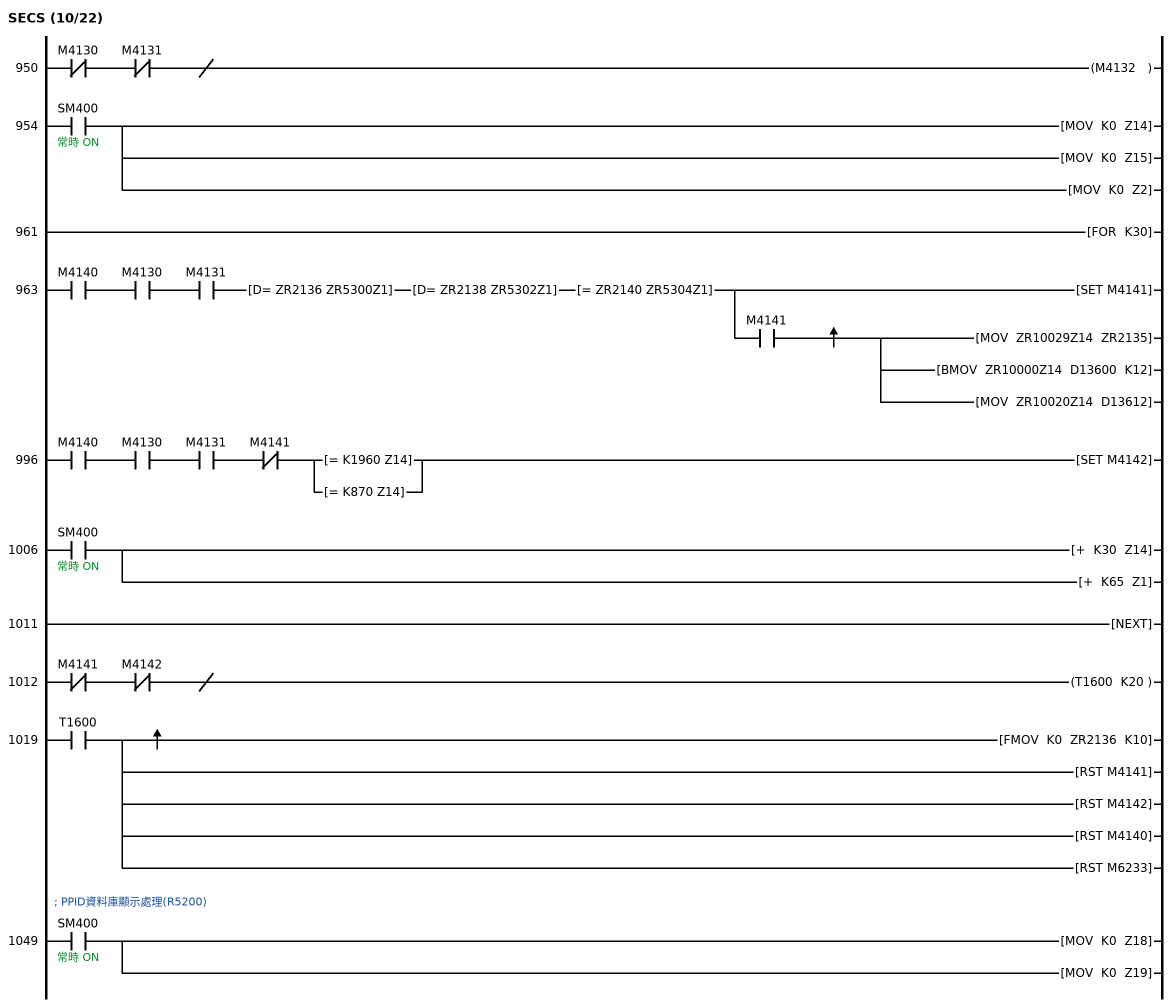
950   LDI     M4130
      ANI     M4131
      INV
      OUT     M4132
954   LD      SM400  ; 常時 ON
      MOV     K0 Z14
      MOV     K0 Z15
      MOV     K0 Z2
961   FOR     K30
963   LD      M4140
      AND     M4130
      AND     M4131
      ANDD=   ZR2136 ZR5300Z1
      ANDD=   ZR2138 ZR5302Z1
      AND=    ZR2140 ZR5304Z1
      SET     M4141
      AND     M4141
      MEP
      MOV     ZR10029Z14 ZR2135
      BMOV    ZR10000Z14 D13600 K12
      MOV     ZR10020Z14 D13612
996   LD      M4140
      AND     M4130
      AND     M4131
      ANI     M4141
      LD=     K1960 Z14
      OR=     K870 Z14
      ANB
      SET     M4142
1006  LD      SM400  ; 常時 ON
      +       K30 Z14
      +       K65 Z1
1011  NEXT
1012  LDI     M4141
      ANI     M4142
      INV
      OUT     T1600 K20
1019  LD      T1600
      MPS
      MEP
      FMOV    K0 ZR2136 K10
      MPP
      RST     M4141
      RST     M4142
      RST     M4140
      RST     M6233
; PPID資料庫顯示處理(R5200)
1049  LD      SM400  ; 常時 ON
      MOV     K0 Z18
      MOV     K0 Z19
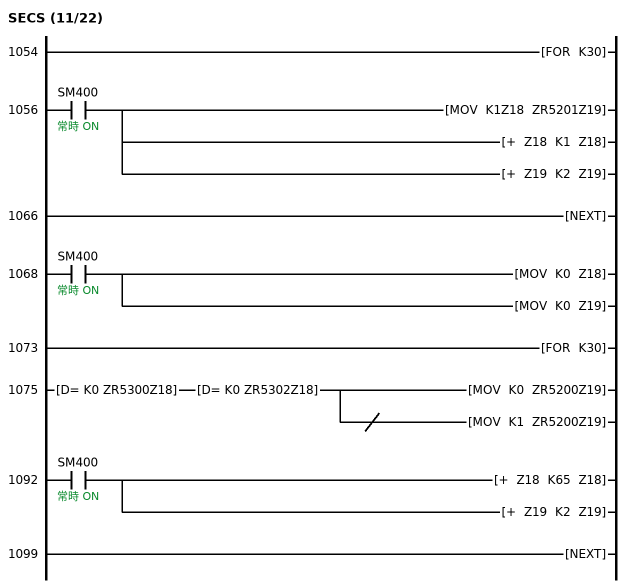
1054  FOR     K30
1056  LD      SM400  ; 常時 ON
      MOV     K1Z18 ZR5201Z19
      +       Z18 K1 Z18
      +       Z19 K2 Z19
1066  NEXT
1068  LD      SM400  ; 常時 ON
      MOV     K0 Z18
      MOV     K0 Z19
1073  FOR     K30
1075  LDD=    K0 ZR5300Z18
      ANDD=   K0 ZR5302Z18
      MOV     K0 ZR5200Z19
      INV
      MOV     K1 ZR5200Z19
1092  LD      SM400  ; 常時 ON
      +       Z18 K65 Z18
      +       Z19 K2 Z19
1099  NEXT
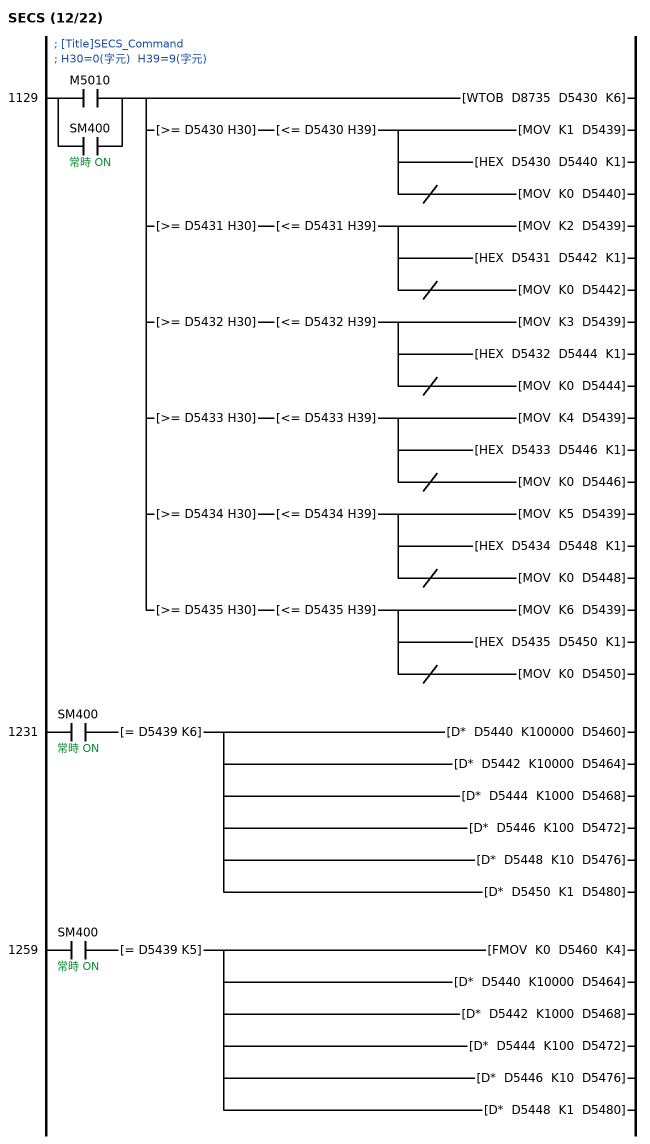
; [Title]SECS_Command
; H30=0(字元)  H39=9(字元)
1129  LD      M5010
      OR      SM400  ; 常時 ON
      WTOB    D8735 D5430 K6
      MPS
      AND>=   D5430 H30
      AND<=   D5430 H39
      MOV     K1 D5439
      HEX     D5430 D5440 K1
      INV
      MOV     K0 D5440
      MRD
      AND>=   D5431 H30
      AND<=   D5431 H39
      MOV     K2 D5439
      HEX     D5431 D5442 K1
      INV
      MOV     K0 D5442
      MRD
      AND>=   D5432 H30
      AND<=   D5432 H39
      MOV     K3 D5439
      HEX     D5432 D5444 K1
      INV
      MOV     K0 D5444
      MRD
      AND>=   D5433 H30
      AND<=   D5433 H39
      MOV     K4 D5439
      HEX     D5433 D5446 K1
      INV
      MOV     K0 D5446
      MRD
      AND>=   D5434 H30
      AND<=   D5434 H39
      MOV     K5 D5439
      HEX     D5434 D5448 K1
      INV
      MOV     K0 D5448
      MPP
      AND>=   D5435 H30
      AND<=   D5435 H39
      MOV     K6 D5439
      HEX     D5435 D5450 K1
      INV
      MOV     K0 D5450
1231  LD      SM400  ; 常時 ON
      AND=    D5439 K6
      D*      D5440 K100000 D5460
      D*      D5442 K10000 D5464
      D*      D5444 K1000 D5468
      D*      D5446 K100 D5472
      D*      D5448 K10 D5476
      D*      D5450 K1 D5480
1259  LD      SM400  ; 常時 ON
      AND=    D5439 K5
      FMOV    K0 D5460 K4
      D*      D5440 K10000 D5464
      D*      D5442 K1000 D5468
      D*      D5444 K100 D5472
      D*      D5446 K10 D5476
      D*      D5448 K1 D5480
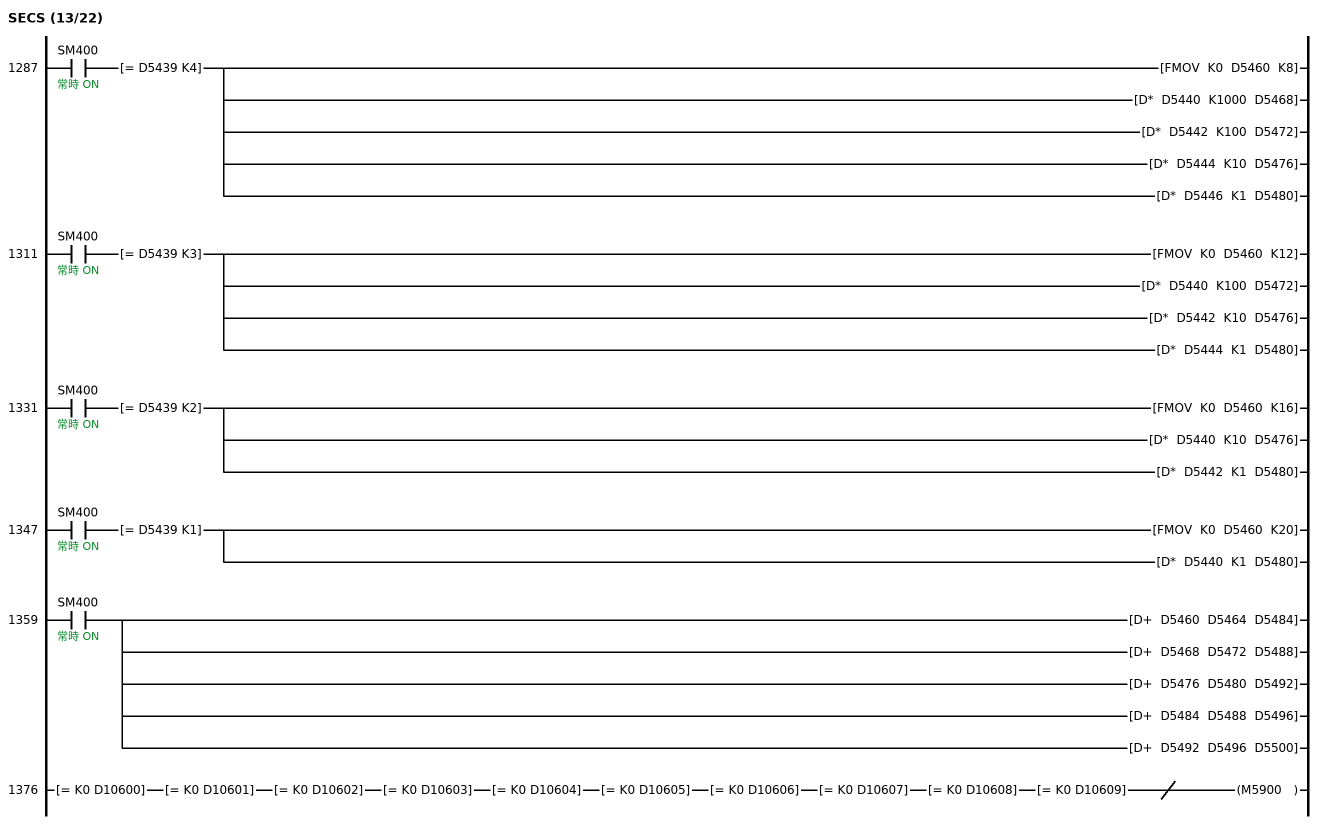
1287  LD      SM400  ; 常時 ON
      AND=    D5439 K4
      FMOV    K0 D5460 K8
      D*      D5440 K1000 D5468
      D*      D5442 K100 D5472
      D*      D5444 K10 D5476
      D*      D5446 K1 D5480
1311  LD      SM400  ; 常時 ON
      AND=    D5439 K3
      FMOV    K0 D5460 K12
      D*      D5440 K100 D5472
      D*      D5442 K10 D5476
      D*      D5444 K1 D5480
1331  LD      SM400  ; 常時 ON
      AND=    D5439 K2
      FMOV    K0 D5460 K16
      D*      D5440 K10 D5476
      D*      D5442 K1 D5480
1347  LD      SM400  ; 常時 ON
      AND=    D5439 K1
      FMOV    K0 D5460 K20
      D*      D5440 K1 D5480
1359  LD      SM400  ; 常時 ON
      D+      D5460 D5464 D5484
      D+      D5468 D5472 D5488
      D+      D5476 D5480 D5492
      D+      D5484 D5488 D5496
      D+      D5492 D5496 D5500
1376  LD=     K0 D10600
      AND=    K0 D10601
      AND=    K0 D10602
      AND=    K0 D10603
      AND=    K0 D10604
      AND=    K0 D10605
      AND=    K0 D10606
      AND=    K0 D10607
      AND=    K0 D10608
      AND=    K0 D10609
      INV
      OUT     M5900
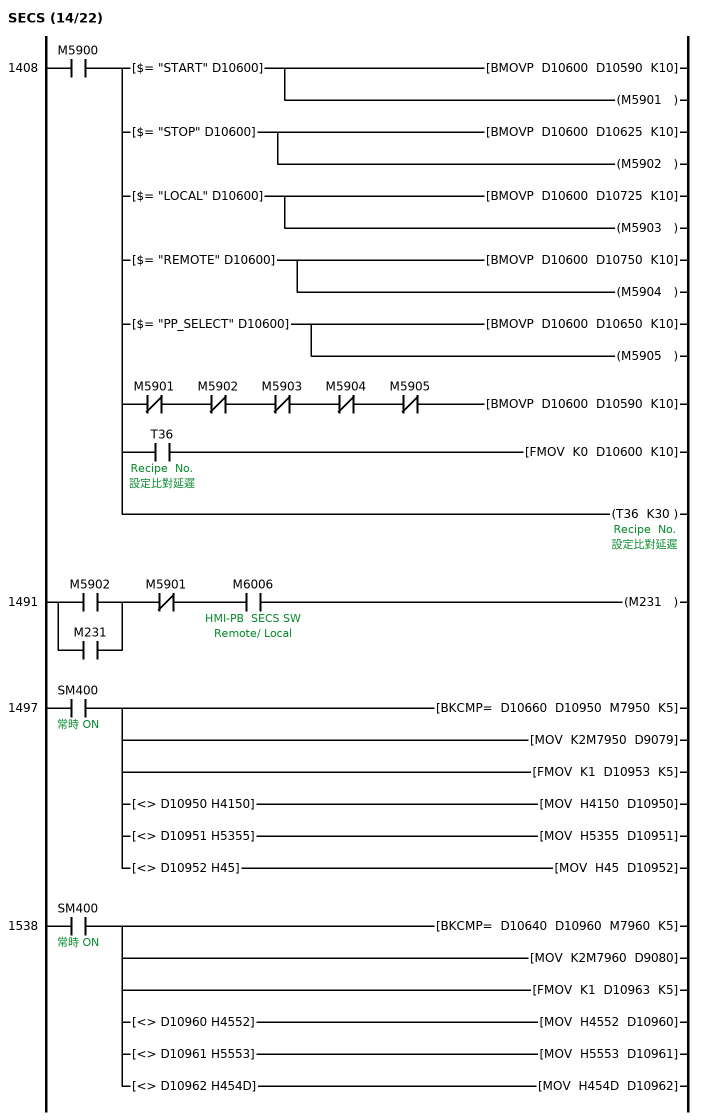
1408  LD      M5900
      MPS
      AND$=   "START" D10600
      BMOVP   D10600 D10590 K10
      OUT     M5901
      MRD
      AND$=   "STOP" D10600
      BMOVP   D10600 D10625 K10
      OUT     M5902
      MRD
      AND$=   "LOCAL" D10600
      BMOVP   D10600 D10725 K10
      OUT     M5903
      MRD
      AND$=   "REMOTE" D10600
      BMOVP   D10600 D10750 K10
      OUT     M5904
      MRD
      AND$=   "PP_SELECT" D10600
      BMOVP   D10600 D10650 K10
      OUT     M5905
      MRD
      ANI     M5901
      ANI     M5902
      ANI     M5903
      ANI     M5904
      ANI     M5905
      BMOVP   D10600 D10590 K10
      MRD
      AND     T36  ; Recipe  No.     設定比對延遲
      FMOV    K0 D10600 K10
      MPP
      OUT     T36 K30  ; Recipe  No.     設定比對延遲
1491  LD      M5902
      OR      M231
      ANI     M5901
      AND     M6006  ; HMI-PB  SECS SW  Remote/ Local
      OUT     M231
1497  LD      SM400  ; 常時 ON
      BKCMP=  D10660 D10950 M7950 K5
        [note] 上位下PAUSE指令
      MOV     K2M7950 D9079
      FMOV    K1 D10953 K5
      MPS
      AND<>   D10950 H4150
      MOV     H4150 D10950
      MRD
      AND<>   D10951 H5355
      MOV     H5355 D10951
      MPP
      AND<>   D10952 H45
      MOV     H45 D10952
1538  LD      SM400  ; 常時 ON
      BKCMP=  D10640 D10960 M7960 K5
        [note] 上位下RESUME指令
      MOV     K2M7960 D9080
      FMOV    K1 D10963 K5
      MPS
      AND<>   D10960 H4552
      MOV     H4552 D10960
      MRD
      AND<>   D10961 H5553
      MOV     H5553 D10961
      MPP
      AND<>   D10962 H454D
      MOV     H454D D10962
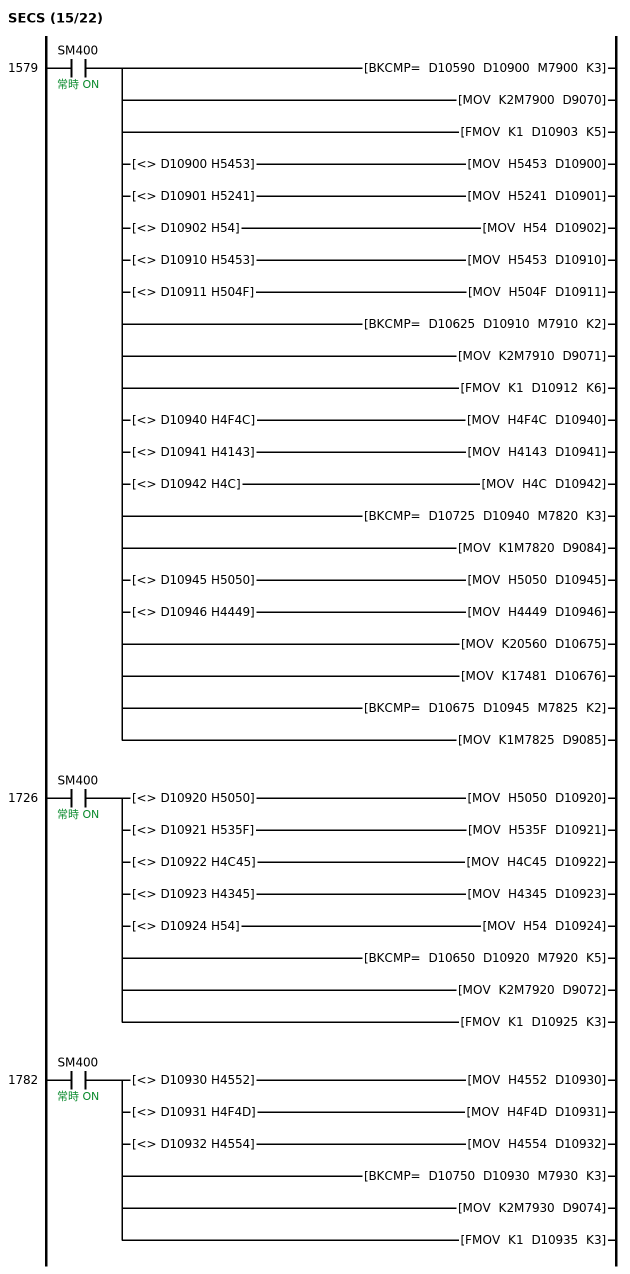
1579  LD      SM400  ; 常時 ON
      BKCMP=  D10590 D10900 M7900 K3
        [note] 上位下START指令
      MOV     K2M7900 D9070
      FMOV    K1 D10903 K5
      MPS
      AND<>   D10900 H5453
      MOV     H5453 D10900
      MRD
      AND<>   D10901 H5241
      MOV     H5241 D10901
      MRD
      AND<>   D10902 H54
      MOV     H54 D10902
      MRD
      AND<>   D10910 H5453
      MOV     H5453 D10910
      MRD
      AND<>   D10911 H504F
      MOV     H504F D10911
      MPP
      BKCMP=  D10625 D10910 M7910 K2
        [note] 上位下STOP指令
      MOV     K2M7910 D9071
      FMOV    K1 D10912 K6
      MPS
      AND<>   D10940 H4F4C
      MOV     H4F4C D10940
      MRD
      AND<>   D10941 H4143
      MOV     H4143 D10941
      MRD
      AND<>   D10942 H4C
      MOV     H4C D10942
      MPP
      BKCMP=  D10725 D10940 M7820 K3
        [note] 上位下GO-LOCAL指令
      MOV     K1M7820 D9084
      MPS
      AND<>   D10945 H5050
      MOV     H5050 D10945
      MRD
      AND<>   D10946 H4449
      MOV     H4449 D10946
      MPP
      MOV     K20560 D10675
      MOV     K17481 D10676
      BKCMP=  D10675 D10945 M7825 K2
        [note] 上位下PPID指令
      MOV     K1M7825 D9085
1726  LD      SM400  ; 常時 ON
      MPS
      AND<>   D10920 H5050
      MOV     H5050 D10920
      MRD
      AND<>   D10921 H535F
      MOV     H535F D10921
      MRD
      AND<>   D10922 H4C45
      MOV     H4C45 D10922
      MRD
      AND<>   D10923 H4345
      MOV     H4345 D10923
      MRD
      AND<>   D10924 H54
      MOV     H54 D10924
      MPP
      BKCMP=  D10650 D10920 M7920 K5
        [note] 上位下PP_SELECT指令
      MOV     K2M7920 D9072
      FMOV    K1 D10925 K3
1782  LD      SM400  ; 常時 ON
      MPS
      AND<>   D10930 H4552
      MOV     H4552 D10930
      MRD
      AND<>   D10931 H4F4D
      MOV     H4F4D D10931
      MRD
      AND<>   D10932 H4554
      MOV     H4554 D10932
      MPP
      BKCMP=  D10750 D10930 M7930 K3
        [note] 上位下GO-REMOTE指令
      MOV     K2M7930 D9074
      FMOV    K1 D10935 K3
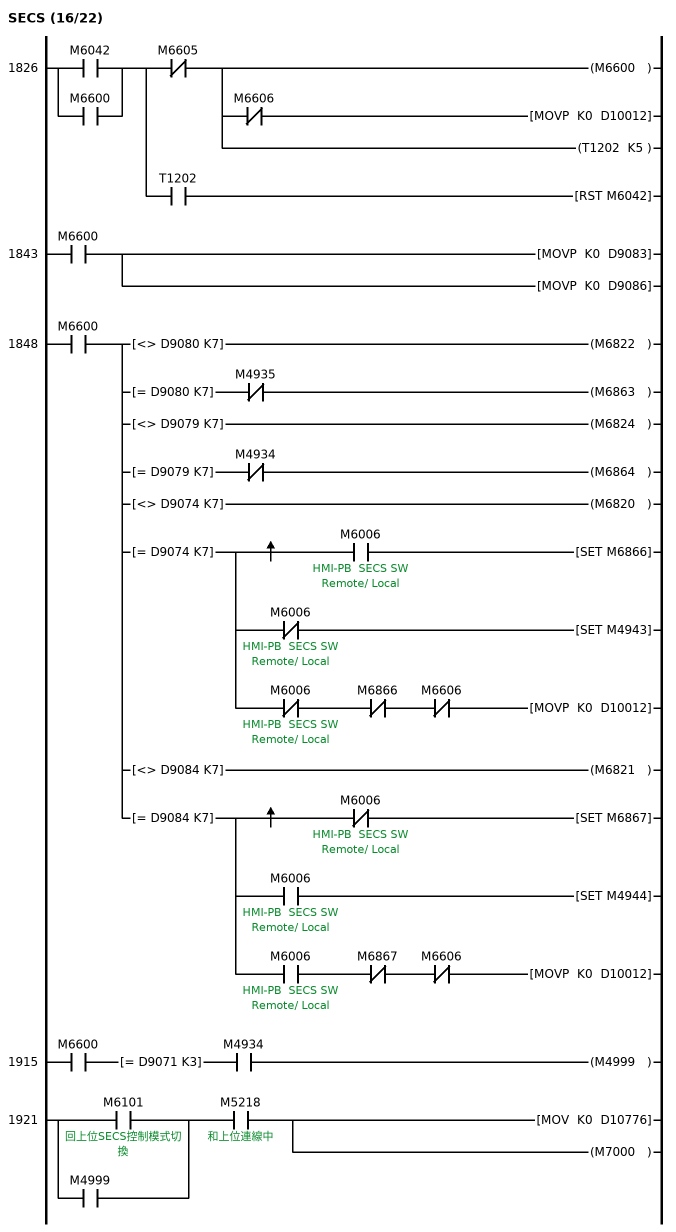
1826  LD      M6042
      OR      M6600
      MPS
      ANI     M6605
      OUT     M6600
      MPS
      ANI     M6606
      MOVP    K0 D10012
      MPP
      OUT     T1202 K5
      MPP
      AND     T1202
      RST     M6042
1843  LD      M6600
      MOVP    K0 D9083
      MOVP    K0 D9086
1848  LD      M6600
      MPS
      AND<>   D9080 K7
      OUT     M6822
      MRD
      AND=    D9080 K7
      ANI     M4935
      OUT     M6863
      MRD
      AND<>   D9079 K7
      OUT     M6824
      MRD
      AND=    D9079 K7
      ANI     M4934
      OUT     M6864
      MRD
      AND<>   D9074 K7
      OUT     M6820
      MRD
      AND=    D9074 K7
      MPS
      MEP
      AND     M6006  ; HMI-PB  SECS SW  Remote/ Local
      SET     M6866
      MRD
      ANI     M6006  ; HMI-PB  SECS SW  Remote/ Local
      SET     M4943
      MPP
      ANI     M6006  ; HMI-PB  SECS SW  Remote/ Local
      ANI     M6866
      ANI     M6606
      MOVP    K0 D10012
      MRD
      AND<>   D9084 K7
      OUT     M6821
      MPP
      AND=    D9084 K7
      MPS
      MEP
      ANI     M6006  ; HMI-PB  SECS SW  Remote/ Local
      SET     M6867
      MRD
      AND     M6006  ; HMI-PB  SECS SW  Remote/ Local
      SET     M4944
      MPP
      AND     M6006  ; HMI-PB  SECS SW  Remote/ Local
      ANI     M6867
      ANI     M6606
      MOVP    K0 D10012
1915  LD      M6600
      AND=    D9071 K3
      AND     M4934
      OUT     M4999
1921  LD      M6101  ; 回上位SECS控制模式切換
      OR      M4999
      AND     M5218  ; 和上位連線中
      MOV     K0 D10776
      OUT     M7000
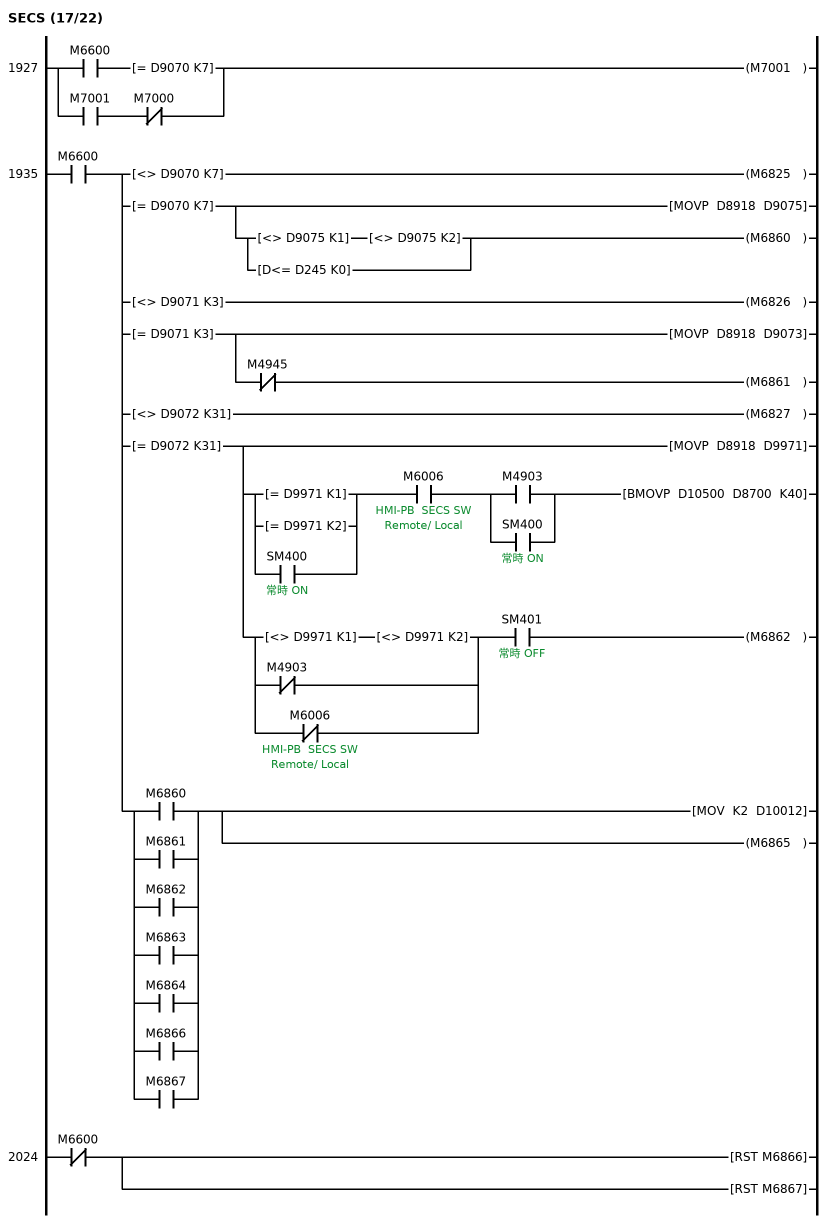
1927  LD      M6600
      AND=    D9070 K7
      LD      M7001
      ANI     M7000
      ORB
      OUT     M7001
1935  LD      M6600
      MPS
      AND<>   D9070 K7
      OUT     M6825
      MRD
      AND=    D9070 K7
      MOVP    D8918 D9075
      LD<>    D9075 K1
      AND<>   D9075 K2
      ORD<=   D245 K0
      ANB
      OUT     M6860
      MRD
      AND<>   D9071 K3
      OUT     M6826
      MRD
      AND=    D9071 K3
      MOVP    D8918 D9073
      ANI     M4945
      OUT     M6861
      MRD
      AND<>   D9072 K31
      OUT     M6827
      MRD
      AND=    D9072 K31
      MOVP    D8918 D9971
      MPS
      LD=     D9971 K1
      OR=     D9971 K2
      OR      SM400  ; 常時 ON
      ANB
      AND     M6006  ; HMI-PB  SECS SW  Remote/ Local
      LD      M4903
      OR      SM400  ; 常時 ON
      ANB
      BMOVP   D10500 D8700 K40
      MPP
      LD<>    D9971 K1
      AND<>   D9971 K2
      ORI     M4903
      ORI     M6006  ; HMI-PB  SECS SW  Remote/ Local
      ANB
      AND     SM401  ; 常時 OFF
      OUT     M6862
      MPP
      LD      M6860
      OR      M6861
      OR      M6862
      OR      M6863
      OR      M6864
      OR      M6866
      OR      M6867
      ANB
      MOV     K2 D10012
      OUT     M6865
2024  LDI     M6600
      RST     M6866
      RST     M6867
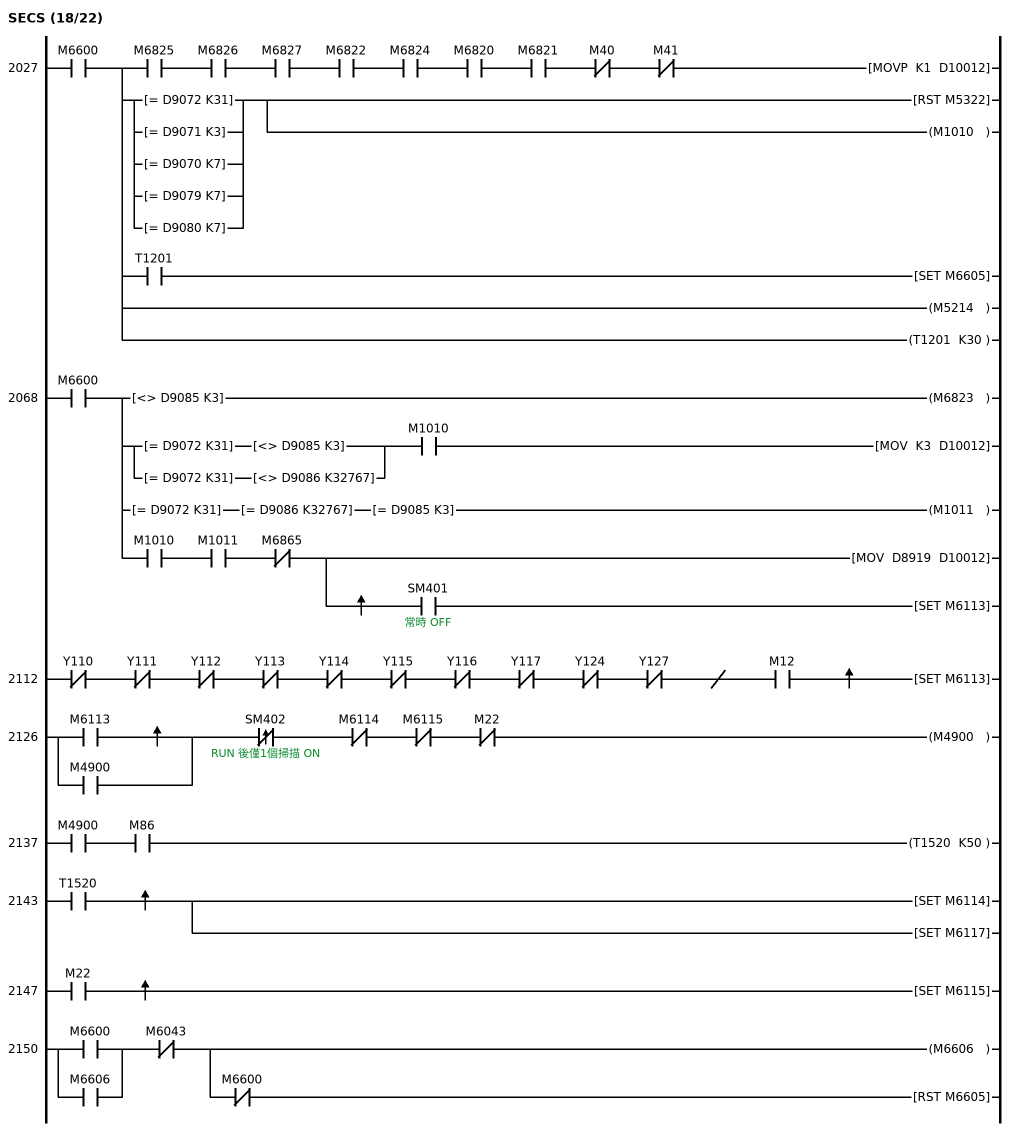
2027  LD      M6600
      MPS
      AND     M6825
      AND     M6826
      AND     M6827
      AND     M6822
      AND     M6824
      AND     M6820
      AND     M6821
      ANI     M40
      ANI     M41
      MOVP    K1 D10012
      MRD
      LD=     D9072 K31
      OR=     D9071 K3
      OR=     D9070 K7
      OR=     D9079 K7
      OR=     D9080 K7
      ANB
      RST     M5322
      OUT     M1010
      MRD
      AND     T1201
      SET     M6605
      MPP
      OUT     M5214
      OUT     T1201 K30
2068  LD      M6600
      MPS
      AND<>   D9085 K3
      OUT     M6823
      MRD
      LD=     D9072 K31
      AND<>   D9085 K3
      LD=     D9072 K31
      AND<>   D9086 K32767
      ORB
      ANB
      AND     M1010
      MOV     K3 D10012
      MRD
      AND=    D9072 K31
      AND=    D9086 K32767
      AND=    D9085 K3
      OUT     M1011
      MPP
      AND     M1010
      AND     M1011
      ANI     M6865
      MOV     D8919 D10012
      MEP
      AND     SM401  ; 常時 OFF
      SET     M6113
2112  LDI     Y110
      ANI     Y111
      ANI     Y112
      ANI     Y113
      ANI     Y114
      ANI     Y115
      ANI     Y116
      ANI     Y117
      ANI     Y124
      ANI     Y127
      INV
      AND     M12
      MEP
      SET     M6113
2126  LD      M6113
      MEP
      OR      M4900
      ANDPI   SM402  ; RUN 後僅1個掃描 ON
      ANI     M6114
      ANI     M6115
      ANI     M22
      OUT     M4900
2137  LD      M4900
      AND     M86
      OUT     T1520 K50
2143  LD      T1520
      MEP
      SET     M6114
      SET     M6117
2147  LD      M22
      MEP
      SET     M6115
2150  LD      M6600
      OR      M6606
      ANI     M6043
      OUT     M6606
      ANI     M6600
      RST     M6605
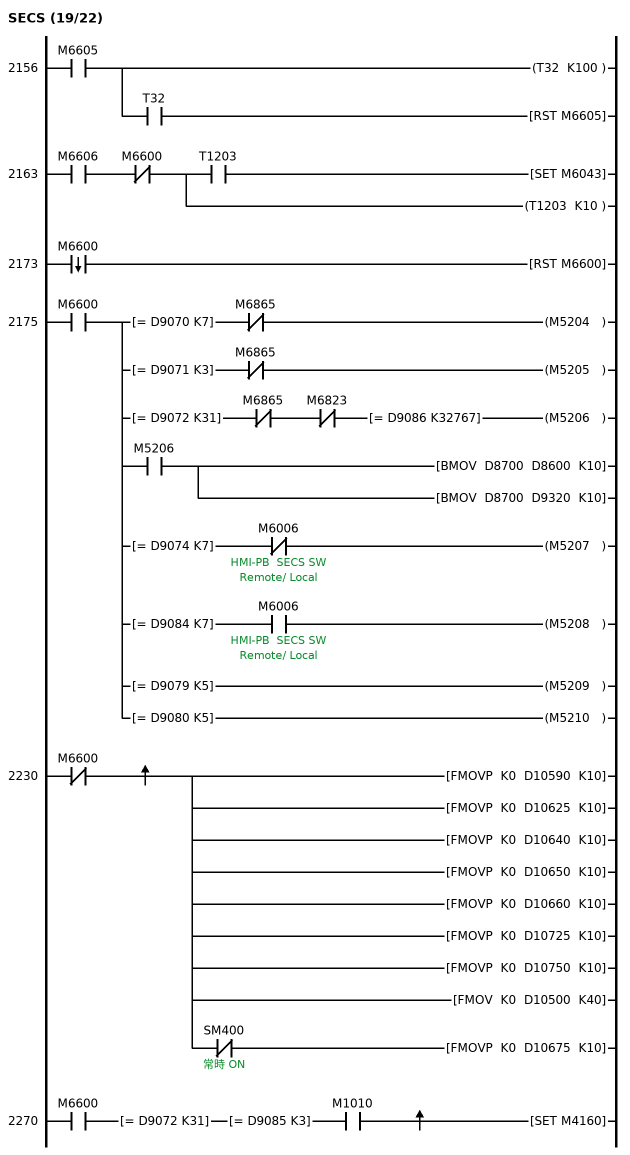
2156  LD      M6605
      OUT     T32 K100
      AND     T32
      RST     M6605
2163  LD      M6606
      ANI     M6600
      MPS
      AND     T1203
      SET     M6043
      MPP
      OUT     T1203 K10
2173  LDF     M6600
      RST     M6600
2175  LD      M6600
      MPS
      AND=    D9070 K7
      ANI     M6865
      OUT     M5204
      MRD
      AND=    D9071 K3
      ANI     M6865
      OUT     M5205
      MRD
      AND=    D9072 K31
      ANI     M6865
      ANI     M6823
      AND=    D9086 K32767
      OUT     M5206
      MRD
      AND     M5206
      BMOV    D8700 D8600 K10
      BMOV    D8700 D9320 K10
      MRD
      AND=    D9074 K7
      ANI     M6006  ; HMI-PB  SECS SW  Remote/ Local
      OUT     M5207
      MRD
      AND=    D9084 K7
      AND     M6006  ; HMI-PB  SECS SW  Remote/ Local
      OUT     M5208
      MRD
      AND=    D9079 K5
      OUT     M5209
      MPP
      AND=    D9080 K5
      OUT     M5210
2230  LDI     M6600
      MEP
      FMOVP   K0 D10590 K10
      FMOVP   K0 D10625 K10
      FMOVP   K0 D10640 K10
      FMOVP   K0 D10650 K10
      FMOVP   K0 D10660 K10
      FMOVP   K0 D10725 K10
      FMOVP   K0 D10750 K10
      FMOV    K0 D10500 K40
      ANI     SM400  ; 常時 ON
      FMOVP   K0 D10675 K10
2270  LD      M6600
      AND=    D9072 K31
      AND=    D9085 K3
      AND     M1010
      MEP
      SET     M4160
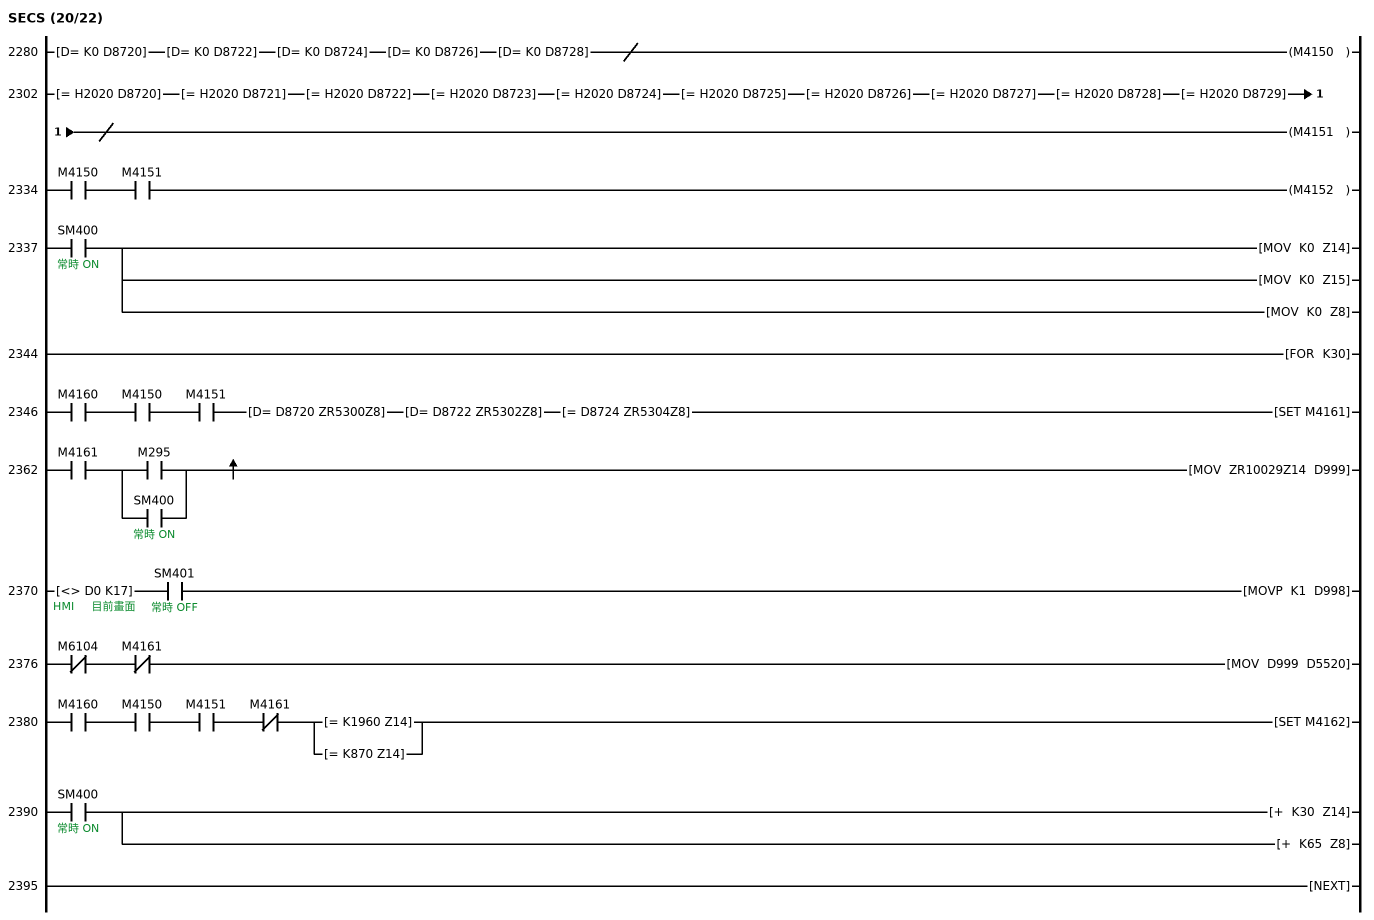
2280  LDD=    K0 D8720
      ANDD=   K0 D8722
      ANDD=   K0 D8724
      ANDD=   K0 D8726
      ANDD=   K0 D8728
      INV
      OUT     M4150
2302  LD=     H2020 D8720
      AND=    H2020 D8721
      AND=    H2020 D8722
      AND=    H2020 D8723
      AND=    H2020 D8724
      AND=    H2020 D8725
      AND=    H2020 D8726
      AND=    H2020 D8727
      AND=    H2020 D8728
      AND=    H2020 D8729
      INV
      OUT     M4151
2334  LD      M4150
      AND     M4151
      OUT     M4152
2337  LD      SM400  ; 常時 ON
      MOV     K0 Z14
      MOV     K0 Z15
      MOV     K0 Z8
2344  FOR     K30
2346  LD      M4160
      AND     M4150
      AND     M4151
      ANDD=   D8720 ZR5300Z8
      ANDD=   D8722 ZR5302Z8
      AND=    D8724 ZR5304Z8
      SET     M4161
2362  LD      M4161
      LD      M295
      OR      SM400  ; 常時 ON
      ANB
      MEP
      MOV     ZR10029Z14 D999
2370  LD<>    D0 K17  ; HMI     目前畫面
      AND     SM401  ; 常時 OFF
      MOVP    K1 D998
2376  LDI     M6104
      ANI     M4161
      MOV     D999 D5520
2380  LD      M4160
      AND     M4150
      AND     M4151
      ANI     M4161
      LD=     K1960 Z14
      OR=     K870 Z14
      ANB
      SET     M4162
2390  LD      SM400  ; 常時 ON
      +       K30 Z14
      +       K65 Z8
2395  NEXT
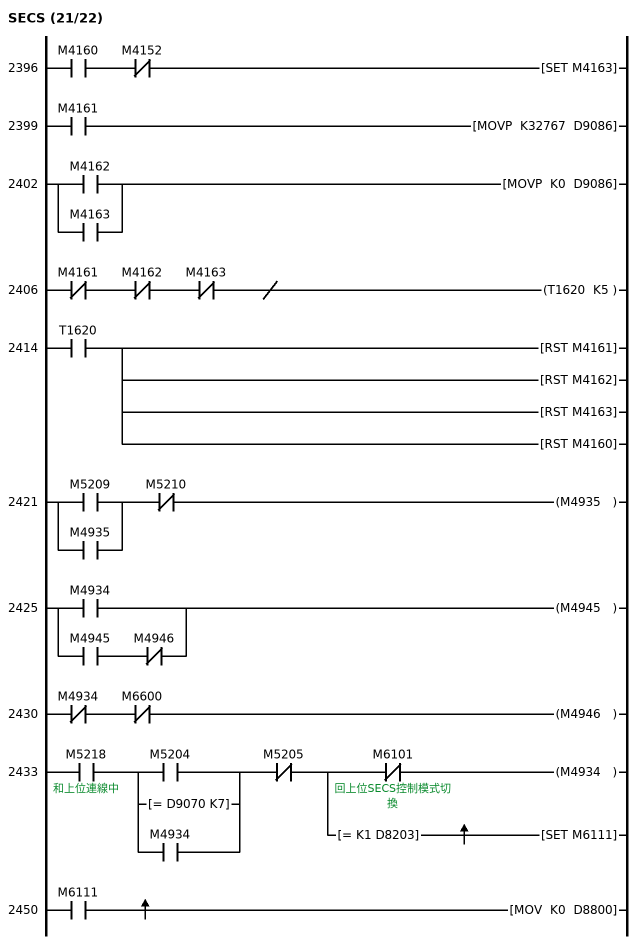
2396  LD      M4160
      ANI     M4152
      SET     M4163
2399  LD      M4161
      MOVP    K32767 D9086
2402  LD      M4162
      OR      M4163
      MOVP    K0 D9086
2406  LDI     M4161
      ANI     M4162
      ANI     M4163
      INV
      OUT     T1620 K5
2414  LD      T1620
      RST     M4161
      RST     M4162
      RST     M4163
      RST     M4160
2421  LD      M5209
      OR      M4935
      ANI     M5210
      OUT     M4935
2425  LD      M4934
      LD      M4945
      ANI     M4946
      ORB
      OUT     M4945
2430  LDI     M4934
      ANI     M6600
      OUT     M4946
2433  LD      M5218  ; 和上位連線中
      LD      M5204
      OR=     D9070 K7
      OR      M4934
      ANB
      ANI     M5205
      MPS
      ANI     M6101  ; 回上位SECS控制模式切換
      OUT     M4934
      MPP
      AND=    K1 D8203
      MEP
      SET     M6111
2450  LD      M6111
      MEP
      MOV     K0 D8800
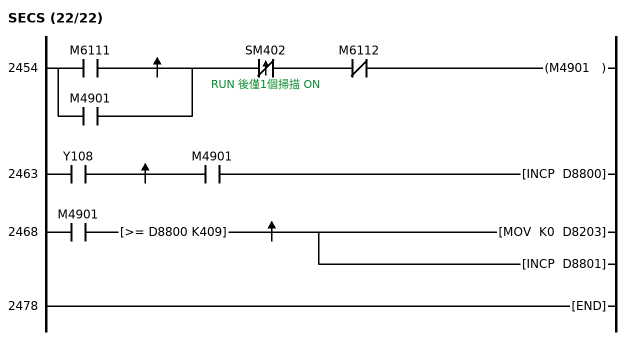
2454  LD      M6111
      MEP
      OR      M4901
      ANDPI   SM402  ; RUN 後僅1個掃描 ON
      ANI     M6112
      OUT     M4901
2463  LD      Y108
      MEP
      AND     M4901
      INCP    D8800
2468  LD      M4901
      AND>=   D8800 K409
      MEP
      MOV     K0 D8203
      INCP    D8801
2478  END
END_PROGRAM

// device comments not shown above
X6  ; 備用
X0C  ; 上游----READY
X0E  ; 下游----READY
Y4B  ; 備用
Y4F  ; 三色燈  藍燈
M505  ; 自動啟動6
M525  ; 自動停止6
T20  ; 開機延遲5s
D301  ; TC01    PV
D302  ; TC02    PV
D350  ; TC01    SV
D351  ; TC02    SV
D601  ; 月 PLC W
D602  ; 日 PLC W
D603  ; 時 PLC W
D604  ; 分 PLC W
D611  ; 月 PLC R
D612  ; 日 PLC R
D613  ; 時 PLC R
D614  ; 分 PLC R
D956  ; 總用電量顯示-1
D957  ; 總用電量顯示-2
D1000  ; RecipeID#02/01
D1016  ; ConveyorSpeed   SV
W0  ; Year    /Month
W1  ; Day  / Hour
W2  ; Min  / Sec
W3  ; / Week
W4  ; Operation Mode
W5  ; Total   WIP     Count
W1A  ; Equipment Status
W1B  ; Alarm/  Warning
W0DC  ; EQP Name#02/#01
W0DD  ; EQP Name#04/#03
W0DE  ; EQP Name#06/#05
W0DF  ; EQP Name#08/#07
W0E0  ; EQP Name#10/#09
W0E1  ; EQP Name#12/#11
W0E2  ; EQP Name#14/#13
W0E3  ; EQP Name#16/#15
W0E4  ; Recipe  No.
W0F7  ; Up      Heat    PV #1
W0F8  ; Up      Heat    PV #2
W0F9  ; Down    Heat    PV #1
W0FA  ; Down    Heat    PV #2
W0FB  ; WIP     Count
W0FC  ; PW      Consump.
W4C5  ; Modify  Type
W4C6  ; Recipe ID #02/#01
W4DA  ; Up-Heat SV
W4DB  ; Down-Heat SV
W4DC  ; Conyeyor Speed
W8C3  ; Index
W0CC2  ; Year    /Month
W0CC3  ; Day  / Hour
W0CC4  ; Min  / Sec
W0CC5  ; / Week
W0CC6  ; HC01    Index
W0CC7  ; Msg     Action
W0D06  ; HC02    Index
W1120  ; Remote  Command
W1600  ; Msg     Action  暫存1
W1601  ; CIM     Message 暫存1
W1640  ; Msg     Action  暫存2
W1680  ; Msg     Action  暫存3
W16C0  ; Msg     Action  暫存4
W1700  ; Msg     Action  暫存1
W1740  ; Msg     Action  暫存2
W1780  ; Msg     Action  暫存3
W17C0  ; Msg     Action  暫存4
W1900  ; Msg     Action  秒數暫存
W1901  ; CIM     Message 暫存#
